PROGRAM SortYourNumbers
VAR
	TestArray : ARRAY[0..9] OF INT := [1,3,8,5,2,9,4,7,6,10];
	SortFinished : BOOL;
	Loop: UINT;
	Temp: INT;
	SwapHappened: BOOL;
END_VAR

//WHILE NOT SortFinished DO
//	IF Loop < ((SIZEOF(TestArray)/2)-1) THEN
//		IF TestArray[Loop] > TestArray[Loop + 1] THEN
//			Temp := TestArray[Loop];
//			TestArray[Loop] := TestArray[Loop + 1];
//			TestArray[Loop + 1] := Temp;
//			SwapHappened := TRUE;
//		END_IF
//		Loop := Loop + 1;
//	ELSE
//		IF SwapHappened THEN
//			SwapHappened := FALSE;
//			Loop := 0;
//		ELSE
//			SortFinished := TRUE;
//		END_IF
//	END_IF
//END_WHILE

AscendingBubbleSort(ArrayToSort := TestArray);

END_PROGRAM

(* stored: Version 1.1.0.1, ProductVersion 3.1.4024.12
   POU SortYourNumbers: Id {1cb95dd3-9e23-406c-9f42-1c70d1bd3662}, SpecialFunc None *)
